// TIA Portal V18 export
FUNCTION "mot_auto_calc_arrived" : Void   // FC17, FBD
{ S7_Optimized_Access := 'TRUE' }
VERSION : 0.1
// stored: AutoNumber true, IsIECCheckEnabled false, SetENOAutomatically false, UDAEnableTagReadback false
   VAR_INPUT
      Target : Real;
      Pos : Real;
      Modifier_delta : Real;
      par_prec_au : Real;
      par_dist_stop : Real;
   END_VAR
   VAR_OUTPUT
      arrived : Bool;
      distance : Real;
      stop_now : Bool;
   END_VAR
BEGIN

REGION Network 2 (SCL)
   #distance := #Target - (#Pos+#Modifier_delta);

   #arrived := ABS(#distance) <= #par_prec_au;

   #stop_now := ABS(#distance) <= #par_dist_stop;
END_REGION
END_FUNCTION
